{attribute 'qualified_only'}
TYPE E_DiffState :
(
    UNKNOWN := 0,
    TRANSFER_ARM_INTERFACE,
    NOMINAL_POSITION
) UINT;
END_TYPE

(* stored: Version 1.1.0.1
   DUT E_DiffState: Id {85889ec6-0695-00d5-2ace-16e5654de6c6} *)
